TYPE E_LockState :
(
	UNDEFINIED,
	Unlocked,
	Locked
)USINT;
END_TYPE

(* stored: Version 1.1.0.1, ProductVersion 3.1.4024.11
   DUT E_LockState: Id {e8deea0b-ea53-47ce-955b-2f3cd9b56598} *)
